Staubli VAL3: __ts_swedish.pgx

program __ts_swedish()
begin
  //
end
